(* IEC 61131-3 sources: plcassist-cli/packages/volt-lsp-iec/test-corpus/bakon-nano/Device/Plc Logic/Application/POUs/LenzeFunctions/EtherCAT, 3 files *)

(* ---- ECAT_MasterHandling.prg ---- *)
PROGRAM ECAT_MasterHandling
(************************************************************)
(* Test EtherCAT libs - ECAT_MasterHandling  	 *)
(************************************************************)
(* Lenze  LAAS-PO 	*)
(************************************************************)
(*   *)
(************************************************************)
(* 1.00	MD				generated  *)

VAR
	xECATRestart			: BOOL;
	SMC3_ReinitAxis_1: L_MC1P_ReinitNode;
	SMC3_ReinitAxis_2: L_MC1P_ReinitNode;
	SMC3_ReinitAxis_3: L_MC1P_ReinitNode;
	SMC3_ReinitAxis_4: L_MC1P_ReinitNode;
	TonRestart : TON;
END_VAR

TonRestart(IN:= g_bResetMaster AND g_HMI_MachCommand.CMD.bResetErrorPulse,PT:=T#0S);
IF TonRestart.Q THEN
	xECATRestart := TRUE;
END_IF

EtherCAT_Master(
	xRestart:= xECATRestart,
	xStopBus:= ,
	xDone=> ,
	xBusy=> ,
	xError=> ,
	eErrorCode=> ,
	wState=> ,
	xDistributedClockInSync=> );

	//EtherCAT_Master.xRestart := xECATRestart;

	SMC3_ReinitAxis_1(
	xExecute:= IoConfig_Globals.EtherCAT_Master.xDone,
	Axis:= IoConfig_Globals.Front_Axis,
	xDone=> ,
	xBusy=> ,
	xError=> ,
	eErrorID=> );

	SMC3_ReinitAxis_2(
	xExecute:= SMC3_ReinitAxis_1.xDone,
	Axis:= IoConfig_Globals.Rear_Axis,
	xDone=> ,
	xBusy=> ,
	xError=> ,
	eErrorID=> );

	SMC3_ReinitAxis_3(
	xExecute:= SMC3_ReinitAxis_2.xDone,
	Axis:= IoConfig_Globals.Z_Axis,
	xDone=> ,
	xBusy=> ,
	xError=> ,
	eErrorID=> );

	SMC3_ReinitAxis_4(
	xExecute:= SMC3_ReinitAxis_3.xDone,
	Axis:= IoConfig_Globals.R_Axis,
	xDone=> ,
	xBusy=> ,
	xError=> ,
	eErrorID=> );

	IF SMC3_ReinitAxis_4.xDone THEN
		xECATRestart := FALSE;
	END_IF

END_PROGRAM

(* ---- Ecat_ReadStatus.prg ---- *)
PROGRAM Ecat_ReadStatus
(************************************************************)
(* Test EtherCAT libs - get  slave state  	 *)
(************************************************************)
(* Lenze  LAAS-PO 	*)
(************************************************************)
(*   *)
(************************************************************)
(* 1.00	FA				generated  *)

VAR
	emd							: L_ETC_DIAGNOSTIC;
	xEcatResetNotifications		: BOOL;
	dwNoOfConfigSlaves			: DWORD;
	dwNoOfConnectedSlaves		: DWORD;

	(* fb instances *)
	ECatMaster					: L_ETC_GetMasterDiagnostic;
	ECatGetSlaveState			: L_ETC_GetSlaveState;

	(* sequence *)
	nSeq							: INT;
	bCyclic							: BOOL:=TRUE;
	wActSlaveAdr					: WORD:=1001;

	(* slave states *)
	wStateTemp					: L_ETC_STATE;
	wStateTemp1					: L_ETC_STATE;
	aEssCur						: ARRAY [1..10] OF L_ETC_STATE ;
	aEssSet						: ARRAY [1..10] OF L_ETC_STATE ;
END_VAR

	ECatMaster(
		xReset:= xEcatResetNotifications,
		xDone=> ,
		xBusy=> ,
		xError=> ,
		eErrorCode=> ,
		oDiagnostic=> emd);

	dwNoOfConfigSlaves := emd.uiNumberOfSlavesConfigured;
	dwNoOfConnectedSlaves := emd.uiNumberOfSlavesFound;

	IF dwNoOfConfigSlaves > 10 THEN
		dwNoOfConfigSlaves := 10;
	END_IF;

	CASE nSeq	OF
	0:
		ECatGetSlaveState(
			xExecute:= TRUE,
			uiDevice:= wActSlaveAdr,
			udiTimeout:= 1000,
			xDone=> ,
			xBusy=> ,
			xError=> ,
			eErrorCode=> ,
			wState=> wStateTemp);

		IF ECatGetSlaveState.xDone OR ECatGetSlaveState.xError THEN
			IF 	NOT ECatGetSlaveState.xError THEN
				(* Uebernahme mit Done, da Zwischenzustaender in der busy-Phase *)
				aEssCur[wActSlaveAdr-1000] := wStateTemp;
				aEssSet[wActSlaveAdr-1000]:= wStateTemp1;
			ELSE
				aEssCur[wActSlaveAdr-1000] := 1;
			END_IF;
			nSeq := 1;
			ECatGetSlaveState(xExecute:= FALSE);
		END_IF;

	1:
		IF wActSlaveAdr >= 1000 + dwNoOfConfigSlaves THEN
			wActSlaveAdr := 1001;
		ELSE
			wActSlaveAdr := wActSlaveAdr +1;
		END_IF;
		nSeq := 2;

	2:
		IF bCyclic THEN
			nSeq := 0;
		END_IF
	END_CASE;

	IF aEssCur[3] = 1 THEN
		g_sMACH.ERR.bErrorComIOStation := TRUE;
	END_IF

	g_bResetMaster := FALSE;
	//FOR i := 1 TO DWORD_TO_INT(dwNoOfConfigSlaves) DO
		IF NOT Front_Axis.xCommunicationOK
			OR NOT Rear_Axis.xCommunicationOK
			OR NOT Z_Axis.xCommunicationOK
			OR NOT R_Axis.xCommunicationOK
			OR g_sMACH.ERR.bErrorComIOStation
			THEN
			g_bResetMaster := TRUE;
		END_IF
	//END_FOR

END_PROGRAM

(* ---- Ecat_SetState.prg ---- *)
PROGRAM Ecat_SetState
(************************************************************)
(* Test EtherCAT libs - set  slave / master state  	 *)
(************************************************************)
(* Lenze  LAAS-PO 	*)
(************************************************************)
(*   *)
(************************************************************)
(* 1.00	FA				generated  *)

VAR
	nSeq				: INT;
	dndummy				: DINT;

	bSetInit			: BOOL;
	bSetPreOP			: BOOL;
	bSetSafeOP			: BOOL;
	bSetOP				: BOOL;

	(* Neuen Status anfordern *)
	wStationAdress		: WORD:=1001;
	esReqState			: L_ETC_STATE :=8;
	bEsSetExec			: BOOL;
	xSetStateDone		: BOOL;
	xSetStateError		: BOOL;

	EcatSetSlaveState	: L_ETC_SetSlaveState;
	sETCerror			: STRING;
	diSetState: INT;
END_VAR

(* check if master is configured *)
IF TRUE THEN

	IF bEsSetExec THEN
		CASE diSetState OF
			0: esReqState :=1;
			1: esReqState :=2;
			2: esReqState :=4;
			3: esReqState :=8;
			ELSE
			esReqState :=8;
		END_CASE
			EcatSetSlaveState(
					xExecute:= TRUE,
					uiDevice:= wStationAdress,
					wState:= esReqState,
					udiTimeout:= 1000,
					xDone=> xSetStateDone,
					xBusy=> ,
					xError=> xSetStateError,
					eErrorCode=> );
			IF EcatSetSlaveState.xError THEN
				sETCerror := L_ETC_GetErrorString( EcatSetSlaveState.eErrorCode, 1);
			END_IF
	ELSE
			sETCerror :=' ';
			IF EcatSetSlaveState.xDone OR EcatSetSlaveState.xError THEN
				EcatSetSlaveState(
					xExecute:= FALSE,
					uiDevice:= wStationAdress,
					wState:= esReqState,
					udiTimeout:= 1000,
					xDone=> xSetStateDone,
					xBusy=> ,
					xError=> xSetStateError,
					eErrorCode=> );
			END_IF;
	END_IF;

END_IF;

END_PROGRAM
